FUNCTION_BLOCK FB_PulseTrigger
VAR_INPUT
	Pulse			:BOOL;
END_VAR
VAR_OUTPUT
	Q				:BOOL;
END_VAR
VAR
	Trigger			:R_Trig; 
	Counter			:INT;
END_VAR

IF Pulse THEN
	Trigger(CLK := TRUE);
ELSE
	Trigger(CLK := FALSE);
END_IF

IF Trigger.Q THEN
	Counter := Counter + 1;
END_IF

IF Counter = 1 THEN
	Q := TRUE;
END_IF
IF Counter = 2 THEN
	Q := FALSE;
	Counter := 0;
END_IF

END_FUNCTION_BLOCK

(* stored: Version 1.1.0.1
   POU FB_PulseTrigger: Id {73d4e208-0771-458b-8770-c4ce372e40a9}, SpecialFunc None *)
